// TIA Portal V17 export
// export: Created 2024-09-02T12:49:57.5741883Z, ExportSetting WithDefaults, DisplayName Totally Integrated Automation Portal, DisplayVersion V17, DisplayName TIA Portal Openness, DisplayVersion V17, DisplayName TIA Portal Version Control Interface, DisplayVersion V17, DisplayName STEP 7 Professional, DisplayVersion V17, DisplayName STEP 7 Safety, DisplayVersion V17, DisplayName WinCC Professional, DisplayVersion V17
FUNCTION "HLP_PosFenster" : Void   // FC30100, LAD
TITLE = Axis position window / Positionsfenster Achse
{ S7_Optimized_Access := 'TRUE' }
AUTHOR : O.Fuehrus
FAMILY : HLP
NAME : HLP
VERSION : 1.0
// stored: AutoNumber false, IsIECCheckEnabled false, SetENOAutomatically false, UDAEnableTagReadback false
   VAR_INPUT
      iFrgInPos : Bool;
      iPosIst : Real;
      iPosSoll : Real;
      iGrenzeMin : Real;
      iGrenzeMax : Real;
   END_VAR
   VAR_OUTPUT
      oInPos : Bool;
      oPosMin : Bool;
      oPosMax : Bool;
   END_VAR
   VAR_TEMP
      t_VKE0 : Bool;   // VKE 0
      t_VKE1 : Bool;   // VKE 1
      tPosMin : Real;
      tPosMax : Real;
   END_VAR
BEGIN

REGION Network 1: VKE0/1
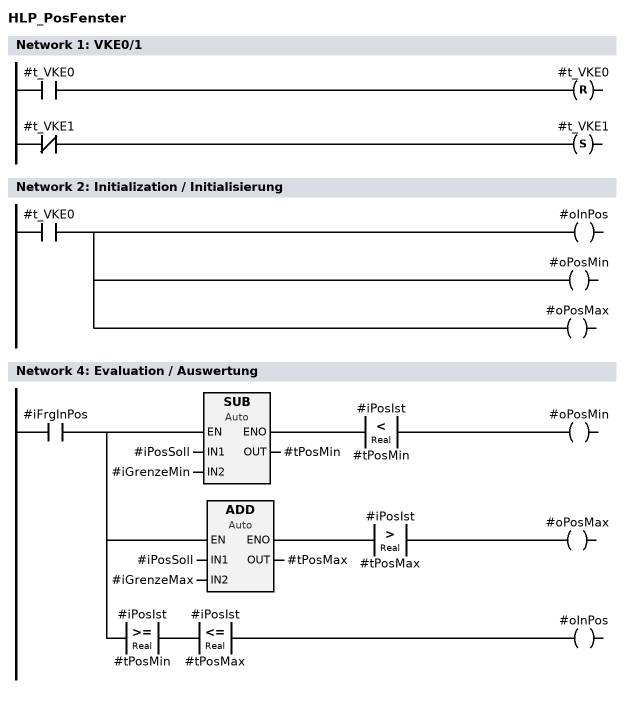
   RUNG wire#powerrail
      Contact( #t_VKE0 )
      R_Coil( #t_VKE0 )
   END_RUNG
   RUNG wire#powerrail
      I_Contact( #t_VKE1 )
      S_Coil( #t_VKE1 )
   END_RUNG
   // the same network as SCL:
   IF #t_VKE0 THEN #t_VKE0 := FALSE; END_IF;
   IF NOT #t_VKE1 THEN #t_VKE1 := TRUE; END_IF;
END_REGION

REGION Network 2: Initialization / Initialisierung
   RUNG wire#powerrail
      Contact( #t_VKE0 )
      wire#w1
      Coil( #oInPos )
   END_RUNG
   RUNG wire#w1
      Coil( #oPosMin )
   END_RUNG
   RUNG wire#w1
      Coil( #oPosMax )
   END_RUNG
   // the same network as SCL:
   #oInPos := #t_VKE0;
   #oPosMin := #t_VKE0;
   #oPosMax := #t_VKE0;
END_REGION

REGION Network 3: Set limits / Grenzen Festlegen
END_REGION

REGION Network 4: Evaluation / Auswertung
   RUNG wire#powerrail
      Contact( #iFrgInPos )
      wire#w1
      Sub(in1 := #iPosSoll, in2 := #iGrenzeMin, out => #tPosMin)
      { S7_Templates := "SrcType := Real" } LT_Contact(in1 := #iPosIst, in2 := #tPosMin)
      Coil( #oPosMin )
   END_RUNG
   RUNG wire#w1
      Add(in1 := #iPosSoll, in2 := #iGrenzeMax, out => #tPosMax)
      { S7_Templates := "SrcType := Real" } GT_Contact(in1 := #iPosIst, in2 := #tPosMax)
      Coil( #oPosMax )
   END_RUNG
   RUNG wire#w1
      { S7_Templates := "SrcType := Real" } GE_Contact(in1 := #iPosIst, in2 := #tPosMin)
      { S7_Templates := "SrcType := Real" } LE_Contact(in1 := #iPosIst, in2 := #tPosMax)
      Coil( #oInPos )
   END_RUNG
   // the same network as SCL:
   IF #iFrgInPos THEN #tPosMin := #iPosSoll - #iGrenzeMin; END_IF;
   #oPosMin := #iFrgInPos AND (#iPosIst < #tPosMin);
   IF #iFrgInPos THEN #tPosMax := #iPosSoll + #iGrenzeMax; END_IF;
   #oPosMax := #iFrgInPos AND (#iPosIst > #tPosMax);
   #oInPos := #iFrgInPos AND (#iPosIst >= #tPosMin) AND (#iPosIst <= #tPosMax);
END_REGION
END_FUNCTION
